TYPE E_DispenserMode :
(
	MODE_None,
	MODE_Piezo,
	MODE_Solenoid
)USINT;
END_TYPE

(* stored: Version 1.1.0.1, ProductVersion 3.1.4022.7
   DUT E_DispenserMode: Id {747323ec-dc12-454f-9769-58fb8244e8f4} *)
